(* PLC project TestProject, CrossPLC TestProject 1.0 *)
(* stored: creationDateTime 2025-09-19T11:56:39, modificationDateTime 2025-09-19T11:56:39 *)

TYPE HMI_UDT : STRUCT
  Start_PB : BOOL;
  Stop_PB : BOOL;
  Start_Active : BOOL;
  Stop_Active : BOOL;
END_STRUCT;
END_TYPE

TYPE P1_UDT : STRUCT
  RW_Tank_tnk_lvl : REAL;
  RW_Pump_flow : REAL;
  RW_Tank_PR_Valve_sts : BOOL;
  RW_Tank_P6B_Valve_sts : BOOL;
  RW_Tank_P_Valve_sts : BOOL;
  RW_Pump_sts : BOOL;
  RW_Pump_fault : BOOL;
  RW_Pump : REAL;
  RW_Tank_PR_Valve : BOOL;
  RW_Tank_P_Valve : BOOL;
  RW_Pump_start : BOOL;
  RW_Pump_stop : BOOL;
  RW_Tank_P6B_Valve : BOOL;
END_STRUCT;
END_TYPE

TYPE P2_UDT : STRUCT
  ChemTreat_NaCl_Tank_tnk_lvl : REAL;
  ChemTreat_NaOCl_Tank_tnk_lvl : REAL;
  ChemTreat_HCl_Tank_tnk_lvl : REAL;
  ChemTreat_NaCl_Tank_Valve_sts : BOOL;
  ChemTreat_NaOCl_Tank_Valve_sts : BOOL;
  ChemTreat_HCl_Tank_Valve_sts : BOOL;
  ChemTreat_NaCl_Tank_Valve : BOOL;
  ChemTreat_NaOCl_Tank_Valve : BOOL;
  ChemTreat_HCl_Tank_Valve : BOOL;
END_STRUCT;
END_TYPE

TYPE P3_UDT : STRUCT
  Ultrafiltration_UFFT_Tank_tnk_lvl : REAL;
  Ultrafiltration_UFFT_Tank_Valve_sts : BOOL;
  Ultrafiltration_UF_Drain_Valve_sts : BOOL;
  Ultrafiltration_UF_ROFT_Valve_sts : BOOL;
  Ultrafiltration_UF_BWP_Valve_sts : BOOL;
  Ultrafiltration_UFFT_Tank_Valve : BOOL;
  Ultrafiltration_UF_Drain_Valve : BOOL;
  Ultrafiltration_UF_ROFT_Valve : BOOL;
  Ultrafiltration_UF_BWP_Valve : BOOL;
END_STRUCT;
END_TYPE

TYPE Phases_UDT : STRUCT
  Filling : BOOL;
  Draining : BOOL;
END_STRUCT;
END_TYPE

TYPE RW_tank_AL_UDT : STRUCT
  LL_alarm : BOOL;
  L_alarm : BOOL;
  H_alarm : BOOL;
  HH_alarm : BOOL;
END_STRUCT;
END_TYPE

TYPE System_State_UDT : STRUCT
  IDLE : BOOL;
  START : BOOL;
  RUNNING : BOOL;
  SHUTDOWN : BOOL;
  Permissives : ARRAY[0..31] OF ?;
  Permissives_Ready : BOOL;
END_STRUCT;
END_TYPE

TYPE SYS_MESSAGES : STRUCT
  ProgramScanTime : DINT;
  AvailableMemory : REAL;
  ControllerStatus : SINT;
  ScanTime : REAL;
END_STRUCT;
END_TYPE

PROGRAM MainProgram
  VAR_INPUT
    Alarms : RW_TANK_AL_UDT;
    GSV_Message : SYS_MESSAGES;
    P1 : P1_UDT;
    P1_SYS : SYSTEM_STATE_UDT;
    P2 : P2_UDT;
    P3 : P3_UDT;
  END_VAR
  VAR_OUTPUT
    HMI : HMI_UDT;
  END_VAR

            (* IO_setup *)
(* P1 Analog Input *)
P1.RW_Tank_tnk_lvl := Local:7:I.Ch0Data;
P1.RW_Pump_flow := Local:7:I.Ch1Data;
(* P1 Digital Input *)
P1.RW_Tank_PR_Valve_sts := Local:2:I.Data.0;
P1.RW_Tank_P6B_Valve_sts := Local:2:I.Data.1;
P1.RW_Tank_P_Valve_sts := Local:2:I.Data.2;
P1.RW_Pump_sts := Local:2:I.Data.3;
P1.RW_Pump_fault := Local:2:I.Data.4;
(* P1 Analog Output *)
P1.RW_Pump := Local:10:O.Ch0Data;
(* Digital Output *)
P1.RW_Tank_PR_Valve := Local:5:O.Data.0;
P1.RW_Tank_P6B_Valve := Local:5:O.Data.1;
P1.RW_Tank_P_Valve := Local:5:O.Data.2;
P1.RW_Pump_start := Local:5:O.Data.3;
P1.RW_Pump_stop := Local:5:O.Data.4;
(* P1 raw water tank alarms *)
Alarms.LL_alarm := Local:7:I.Ch0LLAlarm;
Alarms.L_alarm := Local:7:I.Ch0LAlarm;
Alarms.H_alarm := Local:7:I.Ch0HAlarm;
Alarms.HH_alarm := Local:7:I.Ch0HHAlarm;
(* P2 Analog Input *)
P2.ChemTreat_NaCl_Tank_tnk_lvl := Local:7:I.Ch2Data;
P2.ChemTreat_NaOCl_Tank_tnk_lvl := Local:7:I.Ch3Data;
P2.ChemTreat_HCl_Tank_tnk_lvl := Local:7:I.Ch4Data;
(* P2 Digital Input *)
P2.ChemTreat_NaCl_Tank_Valve_sts := Local:2:I.Data.5;
P2.ChemTreat_NaOCl_Tank_Valve_sts := Local:2:I.Data.6;
(* P2 Analog Output *)
(* NONE *)
(* P2 Digital Output *)
P2.ChemTreat_NaCl_Tank_Valve := Local:5:O.Data.5;
P2.ChemTreat_NaOCl_Tank_Valve := Local:5:O.Data.6;
P2.ChemTreat_HCl_Tank_Valve := Local:5:O.Data.7;
(* P3 Analog Input *)
P3.Ultrafiltration_UFFT_Tank_tnk_lvl := Local:7:I.Ch5Data;
(* P3 Digital Input *)
P3.Ultrafiltration_UFFT_Tank_Valve_sts := Local:2:I.Data.8;
P3.Ultrafiltration_UF_Drain_Valve_sts := Local:2:I.Data.9;
P3.Ultrafiltration_UF_Drain_Valve_sts := Local:2:I.Data.10;
P3.Ultrafiltration_UF_BWP_Valve_sts := Local:2:I.Data.11;
(* P3 Analog Output *)
(* none *)
(* P3 Digital Output *)
P3.Ultrafiltration_UFFT_Tank_Valve := Local:5:O.Data.8;
P3.Ultrafiltration_UF_Drain_Valve := Local:5:O.Data.9;
P3.Ultrafiltration_UF_ROFT_Valve := Local:5:O.Data.10;
P3.Ultrafiltration_UF_BWP_Valve := Local:5:O.Data.11;

(* Raw_water_control *)
P1.RW_Pump_stop := True;
P1.RW_Pump_start := False; (* send the outputs *)
Alarms.LL_alarm := True;
(* if the level is at 500 or lower than 500 open the valve *)
(* output to turn the valve open *)
P1.RW_Tank_PR_Valve := True;
Alarms.L_alarm := True;
(* if level is at 800 *)
P1.RW_Tank_PR_Valve := False; (* close the valve *)
Alarms.H_alarm := True;
Alarms.HH_alarm := True; (* if the tank is higher than or equal to 1200 set the high high alarm *)

(* Raw_water_pump *)
(* start the pump and open the valve from the other tank *)
P1.RW_Tank_P_Valve := True;
P1.RW_Pump_start := True;
P1.RW_Pump_stop := False;
(* stop the pump and close the valve *)
P1.RW_Tank_P_Valve := False;
P1.RW_Pump_stop := True;
P1.RW_Pump_start := False;

(* State_change *)
(* if start and stop is not pressed go to idle *)
P1_SYS.IDLE := True;
P1_SYS.START := False;
P1_SYS.RUNNING := False;
P1_SYS.SHUTDOWN := False;
(* if the start pb and stop is not pressed then change the state of process one to starting *)
P1_SYS.IDLE := False;
P1_SYS.START := True;
P1_SYS.RUNNING := False;
P1_SYS.SHUTDOWN := False;
(* if the tank level is greater than 250 at the start and UFFT is less than a 1000 we can start *)
(* then and all permissves cond together into one tag so we know the plant is ready to start *)
P1_SYS.Permissives_Ready := P1_SYS.Permissives[0] AND P1_SYS.Permissives[1];
(* if the start was pressed and permissives are ready start running Process one *)
P1_SYS.IDLE := False;
P1_SYS.START := False;
P1_SYS.RUNNING := True;
P1_SYS.SHUTDOWN := False;
(* if the stop button is pressed then go to shutdown state *)
P1_SYS.IDLE := False;
P1_SYS.START := False;
P1_SYS.RUNNING := False;
P1_SYS.SHUTDOWN := True;
(* set all permissives to false *)
P1_SYS.Permissives_Ready := False;

          
END_PROGRAM

CONFIGURATION config
  RESOURCE res_MainProgram ON PLC
    TASK task_MainProgram(INTERVAL := T#100ms, PRIORITY := 0);
    PROGRAM MainProgram_instance : MainProgram;
  END_RESOURCE
END_CONFIGURATION
